// TIA Portal project "machTuGiu_setVaReset" (V14)

(* hardware
DEVICE "S7-1200 station_1"  S7-1200 Station
   slot 0: "Rack_0"  S7-1200 Rack  Rack  V1.0
   slot 1: "PLC_1"  CPU 1214C DC/DC/DC  6ES7 214-1AG40-0XB0  V4.2
*)

// ===== PLC "PLC_1"  CPU 1214C DC/DC/DC =====

VAR_GLOBAL   // PLC tag table "Default tag table"
   "Tag_1" AT %I0.0 : Bool;
   "Tag_2" AT %Q0.0 : Bool;
   "Tag_3" AT %I0.1 : Bool;
   "Tag_4" AT %I0.2 : Bool;
   "Tag_5" AT %Q0.1 : Bool;
   "Tag_6" AT %Q0.2 : Bool;
   "Tag_7" AT %I0.3 : Bool;
   "Tag_8" AT %Q0.3 : Bool;
END_VAR

ORGANIZATION_BLOCK "Main"   // OB1, LAD, ProgramCycle
TITLE = "Main Program Sweep (Cycle)"
{ S7_Optimized_Access := 'TRUE' }
VERSION : 0.1
   VAR_INPUT
      Initial_Call : Bool;   // Initial call of this OB
      Remanence : Bool;   // =True, if remanent data are available
   END_VAR
BEGIN

REGION Network 1
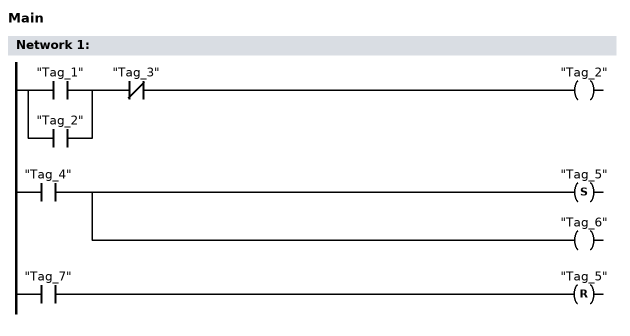
   RUNG wire#powerrail
      Contact( "Tag_1" )
      wire#w1
      I_Contact( "Tag_3" )
      Coil( "Tag_2" )
   END_RUNG
   RUNG wire#powerrail
      Contact( "Tag_2" )
   END_RUNG wire#w1
   RUNG wire#powerrail
      Contact( "Tag_4" )
      wire#w2
      S_Coil( "Tag_5" )
   END_RUNG
   RUNG wire#w2
      Coil( "Tag_6" )
   END_RUNG
   RUNG wire#powerrail
      Contact( "Tag_7" )
      R_Coil( "Tag_5" )
   END_RUNG
   // the same network as SCL:
   "Tag_2" := ("Tag_1" OR "Tag_2") AND NOT "Tag_3";
   IF "Tag_4" THEN "Tag_5" := TRUE; END_IF;
   "Tag_6" := "Tag_4";
   IF "Tag_7" THEN "Tag_5" := FALSE; END_IF;
END_REGION
END_ORGANIZATION_BLOCK